{attribute 'qualified_only'}
VAR_GLOBAL
	
PRESSURE_SENSE AT %I*:BOOL;
HUM_SENS,HUM_SENS2 AT %I*:INT;


ENABLE AT %Q*:BOOL;
FL1,FL2,FL3 AT %Q*:BOOL;
INCAN AT %Q*:INT;
//HPS1,HPS2,HPS3 AT %Q*:BOOL; //Not used in TCR120

AUX1,AUX2,AUX3,ALARM AT %Q*:BOOL; 
HEATERS AT %Q*:BOOL;

HUMVALVE AT %Q*:BOOL;

GLYCOL_VALVE AT %Q*:INT;

END_VAR

VAR_GLOBAL PERSISTENT
	FANSPEED AT %Q*:INT;
END_VAR

(* stored: Version 1.1.0.1, ProductVersion 3.1.4022.18
   GVL IO_VARS: Id {5deb4137-ac2e-40b5-80c9-14b62d0f5cec} *)
